# EPICS autosave request: iocBoot/sioc-gunb-fc01/sioc-gunb-fc01.req
file "kiethly.req" AREA=GUNB,POS=753
